VAR_GLOBAL PERSISTENT
	
/////////////////////////////////////////////////////////////////////////////////////Log/////////////////////////////////////////////////////////////////////////////////////
	
	stUserLog					: ARRAY [0..250] OF ST_UserLog;
	
	aDataHistoryNest1			: ARRAY[0..2000] OF ST_CycleData;
	aDataHistoryNest2			: ARRAY[0..2000] OF ST_CycleData;
	astEventsHistory			: ARRAY[0..200] OF ST_EventsHistory;

	lastDateCSV					: STRING;

END_VAR

(* stored: Version 1.1.0.1, ProductVersion 3.1.4026.18
   GVL GVL_Persistent: Id {c4d03ea6-35af-4633-972d-fef3cfe7daa9} *)
